PROGRAM MAIN
VAR
END_VAR

END_PROGRAM

(* stored: Version 1.1.0.1
   POU MAIN: Id {dae7e471-9550-49b5-82fe-caf6bfedea2d} *)
